// TwinCAT 3 PLC project PLC_1
// ProgramVersion: 3.1.4023.0
// libraries:
//   Tc2_Standard, * (Beckhoff Automation GmbH)
//   Tc2_System, * (Beckhoff Automation GmbH)
//   Tc2_Utilities, * (Beckhoff Automation GmbH)
//   Tc3_Module, * (Beckhoff Automation GmbH)
// project tree:
//   / PlcTask.TcTTO
//   POUs/ MAIN.TcPOU

CONFIGURATION PLC_1
    RESOURCE PLC ON TwinCAT3
        TASK PlcTask(INTERVAL := T#10ms, PRIORITY := 20);
        PROGRAM MAIN WITH PlcTask : MAIN;
    END_RESOURCE
END_CONFIGURATION

// ---- POUs/MAIN.TcPOU
PROGRAM MAIN
VAR
	ntGetTime	: NT_GetTime;
	timeST		: Tc2_Utilities.TIMESTRUCT;
	
	ton			: TON;
	
	fbLocalSystemTime	: FB_LocalSystemTime;
END_VAR

ton(IN := NOT ton.Q, PT := T#100MS);

ntGetTime(
	NETID := '26.242.21.199.1.1',
	START := ton.Q,
	TIMESTR => timeST);
	
fbLocalSystemTime(
	sNetID:= '', 
	bEnable:= TRUE);

END_PROGRAM
